PROGRAM POU
VAR
	running: BOOL;
	currentError: UDINT;
	done: BOOL;
	busy: BOOL;
	reset: BOOL;
	position: LREAL;
END_VAR

HAVL.axis.ReadStatus();

HAVL.axisPower(
	Axis:= HAVL.axis,
	Enable:= HAVL.enable,
	Enable_Positive:= HAVL.enable,
	Enable_Negative:= HAVL.enable,
	Override:= HAVL.override,
	BufferMode:= ,
	Options:= ,
	Status=> running,
	Busy=> ,
	Active=> ,
	Error=> ,
	ErrorID=> currentError
);

HAVL.axisMoveAbsolute(
	Axis:= HAVL.axis,
	Execute:= HAVL.enableMove,
	Position:= HAVL.targetPosition,
	Velocity:= HAVL.targetVelocity,
	Acceleration:= ,
	Deceleration:= ,
	Jerk:= ,
	BufferMode:= ,
	Options:= ,
	Done=> done,
	Busy=> busy,
	Active=> ,
	CommandAborted=> ,
	Error=> ,
	ErrorID=> currentError 
);

HAVL.axisErrorReset(Axis := HAVL.axis, Execute := reset, Done =>, Error =>, ErrorID => currentError);

HAVL.axisReadActualPosition(Axis := HAVL.axis, Enable := busy, Valid=>, Busy=>, Error=>, ErrorID=>, Position=> position);

END_PROGRAM

(* stored: Version 1.1.0.1, ProductVersion 3.1.4024.6
   POU POU: Id {432c7f74-8b66-4450-8a66-d7a918564091}, SpecialFunc None *)
